# EPICS autosave request: iocBoot/iocSR06IOC01/SR06IOC01_DMC01Positions.req
$(P)A.DVAL
$(P)B.DVAL
$(P)C.DVAL
$(P)D.DVAL
